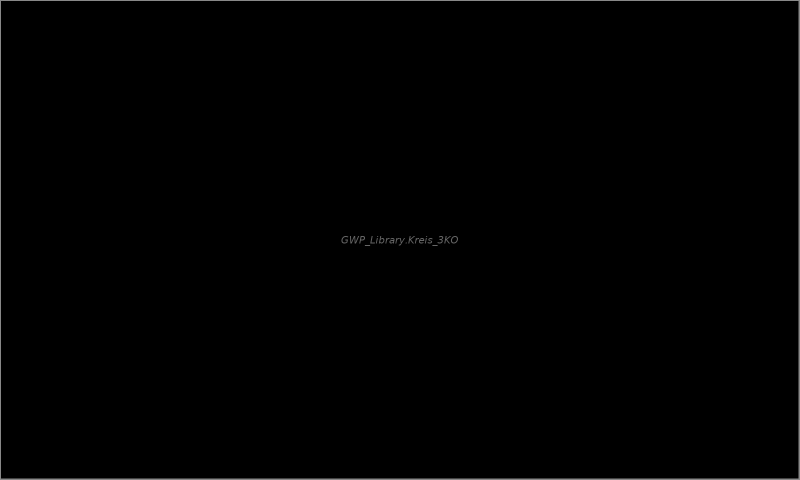
VISUALIZATION Kreis  // 800x480
    Frame (0,0 800x480)
        shows GWP_Library.Kreis_3KO(FB_Kreis_3KO := MAIN.Kreis_3KO_0, FB_KD := MAIN.KD_0, FB_VD := MAIN.VD_0, FB_Init_1 := MAIN.Init_0)
END_VISUALIZATION

(* stored: Version 1.1.0.1, ProductVersion 3.1.4022.6
   Visu Kreis: Id {61e92546-efaa-4641-baf1-b7b3397efa66} *)
